FUNCTION_BLOCK Z2 
VAR_INPUT	
	ENABLE     : BOOL;
	EMG        : BOOL;
	RIPRISTINO : BOOL;
	LIBERO_I   : BOOL;
	TRIGGER_I  : BOOL;
a_0 : BOOL;
a_1	: BOOL;
I5 : BOOL;

END_VAR
VAR_OUTPUT
LIBERO_O   : BOOL;
TRIGGER_O  : BOOL;	
Q1 : BOOL;
Q2 : BOOL;

END_VAR

VAR	
stato : (S_attesa, S_uscita, S_Rientro, S_Ripristino, S_Emergenza) := S_attesa;
S_attesa : BOOL;
S_Uscita : BOOL;
S_rientro : BOOL;
S_ripristino : BOOL;
S_emergenza  : BOOL;
Trigger_OUT : TON();

END_VAR

//dichiarazione timer

Trigger_OUT(IN := Trigger_OUT.Q, PT := T#3S);

//Comandi transizione degli stati


IF EMG = FALSE  OR Enable = FALSE THEN
	
	stato := S_Emergenza;
	
END_IF

CASE stato OF
	S_Emergenza:
	
		IF Enable = TRUE AND Ripristino = TRUE THEN
		
			stato := S_Ripristino;
		
		END_IF
		
		Q1 := FALSE;
		Q2 := FALSE;
		Libero_O := FALSE;
		Trigger_O := FALSE;
	S_Ripristino:
		
		IF Enable = TRUE AND a_0 = TRUE THEN
			
			stato := S_Attesa;
			
		END_IF
		
		Q1 := TRUE;
		Q2 := FALSE;
		libero_O := FALSE;
		Trigger_O := FALSE;
	
	S_Attesa: 
	
		IF Enable = TRUE AND Trigger_I = TRUE AND Libero_I = TRUE AND a_0 = TRUE THEN
			
			stato := S_Uscita;
			
		END_IF
	
		Q1 := FALSE;
		Q2 := FALSE;
		Libero_O := TRUE;
		Trigger_O := FALSE;
	S_Uscita:
	
		IF a_1 = TRUE THEN
			
			stato := S_Rientro;
			
		END_IF
	
		Q1 := FALSE;
		Q2 := TRUE;
		Libero_O := FALSE;
		Trigger_O := FALSE;
	
S_Rientro:
	
		IF a_0 = TRUE THEN
			
			stato := S_Attesa;
			
		END_IF
	
		Q1 := TRUE;
		Q2 := FALSE;
		Libero_O := TRUE;
		Trigger_OUT.Q;
		Trigger_O := TRUE;
END_CASE

END_FUNCTION_BLOCK

(* stored: Version 1.1.0.1, ProductVersion 3.1.4024.12
   POU Z2: Id {6dde8437-606b-4d0e-8b96-5f698fbf635a}, SpecialFunc None *)
